(*
SPDX-FileCopyrightText: © 2026 Oleksandr Tiutyk <trofimich@gmail.com>
SPDX-License-Identifier: MIT
License: https://opensource.org/license/mit
*)

(*!
<summary>
Beckhoff EL4008: 8-channel analog output terminal (0 .. 10 V, 12-bit).
</summary>
<description>
Process image mapping structure for the EL4008 EtherCAT terminal with 8 analog output channels (0 .. 10 V,
12-bit).
When used for I/O, link located fields or their containing buffers to the matching selected PDOs.
The record is not a packed wire buffer; compiler padding is not part of the device specification.
Unlinked/default values do not prove valid I/O. The caller evaluates bus/channel validity before use.
Use one owner task per instance and externally synchronize other access; multi-field snapshots are not atomic.
Copies store data without creating hardware links. Keep borrowed field references valid while consumers are bound.
This passive record performs no validation, synchronization, configuration or protocol advancement.
Channels hold raw INT16 output commands; configure electrical range and presentation before use.
</description>
*)
TYPE EL4008 :
STRUCT
	Ch1 AT %Q* : INT;
	Ch2 AT %Q* : INT;
	Ch3 AT %Q* : INT;
	Ch4 AT %Q* : INT;
	Ch5 AT %Q* : INT;
	Ch6 AT %Q* : INT;
	Ch7 AT %Q* : INT;
	Ch8 AT %Q* : INT;
END_STRUCT
END_TYPE

(* stored: Version 1.1.0.1, ProductVersion 3.1.4026.20
   DUT EL4008: Id {7cf8b8d6-2e13-48ee-867c-8a8556f97183} *)
